PROGRAM MAIN
VAR
END_VAR

END_PROGRAM

(* stored: Version 1.1.0.1
   POU MAIN: Id {63912e07-ae13-4c1c-baba-4d0bcf96ddff} *)
